// TIA Portal project "tram_2_full_V16" (V16)

(* hardware
DEVICE "S7-1200 station_1"  S7-1200 Station
   slot 0: "Rack_0"  S7-1200 Rack  Rack  V1.0
   slot 1: "PLC_1"  CPU 1214C DC/DC/DC  6ES7 214-1AG40-0XB0  V4.1
   slot 2: "DQ 8xRelay_1"  SM 1222 DQ8 x relay  6ES7 222-1HF32-0XB0  V2.0
DEVICE "HMI_1"  KTP400 Basic PN
   slot 0: "HMI_1"  KTP400 Basic PN  6AV2 123-2DB03-0AX0  15.0.0.0
   slot 1: "HMI_RT_1"  KTP400 Basic PN  6AV2 123-2DB03-0AX0  15.0.0.0
   slot 5: "HMI_1.IE_CP_1"  PROFINET Interface  15.0.0.0
      slot 1: "PROFINET Interface_1"  PROFINET Interface
         slot 1: "Port_1"  Port
*)

// ===== PLC "PLC_1"  CPU 1214C DC/DC/DC =====

VAR_GLOBAL   // PLC tag table "Default tag table"
   "Start" AT %I0.1 : Bool;
   "CylinderB" AT %Q9.6 : Bool;
   "Gripper" AT %Q9.5 : Bool;
   "Arm+" AT %Q9.4 : Bool;
   "Stop" AT %I0.2 : Bool;
   "Arm-" AT %Q9.3 : Bool;
   "CylinderA-" AT %Q9.2 : Bool;
   "CylinderA+" AT %Q9.7 : Bool;
   "Tag_1" AT %M0.1 : Bool;
   "Timer1" AT %MD0 : DWord;
   "LQ2" AT %I0.6 : Bool;
   "SQ3" AT %I0.7 : Bool;
   "Tag_2" AT %M0.2 : Bool;
   "Timer2" AT %MD4 : DWord;
   "Tag_3" AT %M0.3 : Bool;
   "Tag_4" AT %M0.4 : Bool;
   "Tag_5" AT %M1.1 : Bool;
   "Tag_6" AT %M0.7 : Bool;
   "Tag_7" AT %M1.4 : Bool;
   "LQ1" AT %I0.5 : Bool;
   "Tag_8" AT %Q9.0 : Bool;
   "Tag_9" AT %Q9.1 : Bool;
   "Timer4" AT %MD10 : DWord;
   "Timer5" AT %MD14 : DWord;
   "Tag_10" AT %Q0.1 : Bool;
   "Tag_11" AT %Q0.2 : Bool;
   "Tag_12" AT %M0.5 : Bool;
   "MemoryStop" AT %Q0.3 : Bool;
   "Tag_13" AT %Q0.4 : Bool;
   "Tag_14" AT %M4.5 : Bool;
END_VAR

// folder: System blocks/Program resources

DATA_BLOCK "T1"   // DB1
{ S7_Optimized_Access := 'TRUE' }
AUTHOR : Simatic
FAMILY : IEC
NAME : IEC_TMR
VERSION : 1.0
// stored: InstanceOfName IEC_TIMER
"IEC_TIMER"
BEGIN
END_DATA_BLOCK

DATA_BLOCK "T4"   // DB3
{ S7_Optimized_Access := 'TRUE' }
AUTHOR : Simatic
FAMILY : IEC
NAME : IEC_TMR
VERSION : 1.0
// stored: InstanceOfName IEC_TIMER
"IEC_TIMER"
BEGIN
END_DATA_BLOCK

// folder: (top level)

ORGANIZATION_BLOCK "Main"   // OB1, LAD, ProgramCycle
TITLE = "Main Program Sweep (Cycle)"
{ S7_Optimized_Access := 'TRUE' }
VERSION : 0.1
   VAR_INPUT
      Initial_Call : Bool;   // Initial call of this OB
      Remanence : Bool;   // =True, if remanent data are available
   END_VAR
   VAR_TEMP   // added for the SCL form of the ladder/FBD networks
      _w1 : Bool;
   END_VAR
BEGIN

REGION Network 1
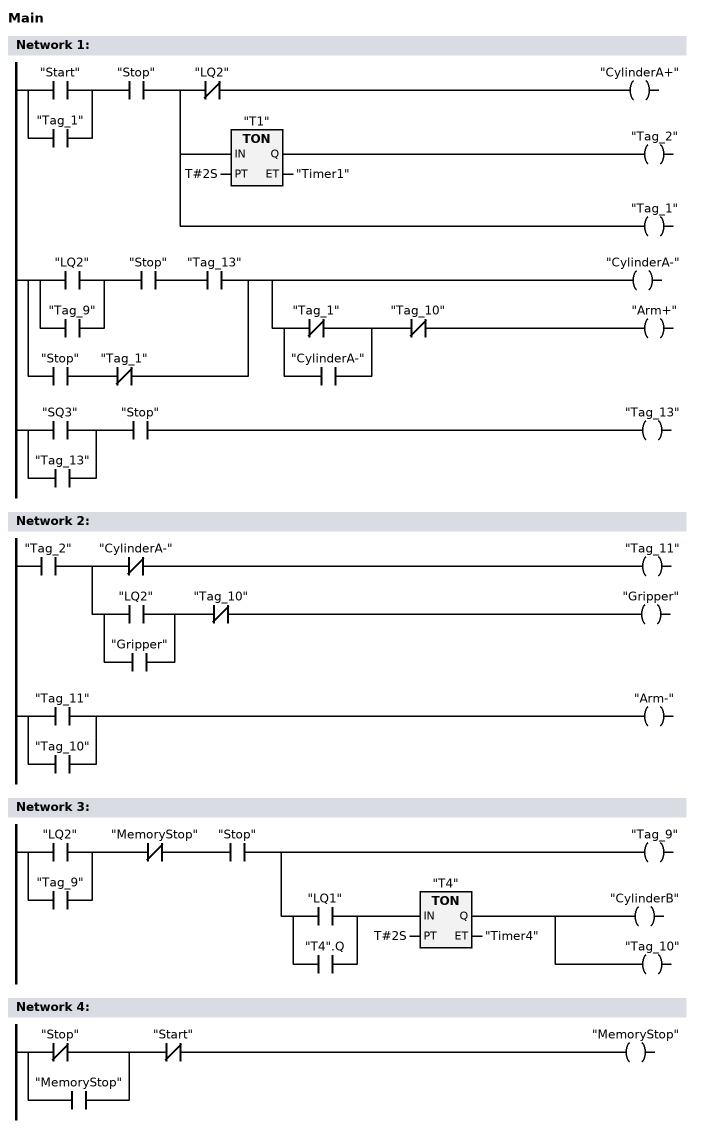
   #_w1 := ("Start" OR "Tag_1") AND "Stop";
   "CylinderA+" := #_w1 AND NOT "LQ2";
   "T1".TON(IN := #_w1, PT := T#2S, ET => "Timer1");
   "Tag_2" := "T1".Q;
   "Tag_1" := #_w1;
   "CylinderA-" := (("LQ2" OR "Tag_9") AND "Stop" AND "Tag_13") OR ("Stop" AND NOT "Tag_1");
   "Arm+" := "CylinderA-" AND (NOT "Tag_1" OR "CylinderA-") AND NOT "Tag_10";
   "Tag_13" := ("SQ3" OR "Tag_13") AND "Stop";
END_REGION

REGION Network 2
   RUNG wire#powerrail
      Contact( "Tag_2" )
      wire#w1
      I_Contact( "CylinderA-" )
      Coil( "Tag_11" )
   END_RUNG
   RUNG wire#w1
      Contact( "LQ2" )
      wire#w2
      I_Contact( "Tag_10" )
      Coil( "Gripper" )
   END_RUNG
   RUNG wire#w1
      Contact( "Gripper" )
   END_RUNG wire#w2
   RUNG wire#powerrail
      Contact( "Tag_11" )
      wire#w3
      Coil( "Arm-" )
   END_RUNG
   RUNG wire#powerrail
      Contact( "Tag_10" )
   END_RUNG wire#w3
   // the same network as SCL:
   "Tag_11" := "Tag_2" AND NOT "CylinderA-";
   "Gripper" := "Tag_2" AND ("LQ2" OR "Gripper") AND NOT "Tag_10";
   "Arm-" := "Tag_11" OR "Tag_10";
END_REGION

REGION Network 3
   "Tag_9" := ("LQ2" OR "Tag_9") AND NOT "MemoryStop" AND "Stop";
   "T4".TON(IN := "Tag_9" AND ("LQ1" OR "T4".Q), PT := T#2S, ET => "Timer4");
   "CylinderB" := "T4".Q;
   "Tag_10" := "T4".Q;
END_REGION

REGION Network 4
   RUNG wire#powerrail
      I_Contact( "Stop" )
      wire#w1
      I_Contact( "Start" )
      Coil( "MemoryStop" )
   END_RUNG
   RUNG wire#powerrail
      Contact( "MemoryStop" )
   END_RUNG wire#w1
   // the same network as SCL:
   "MemoryStop" := (NOT "Stop" OR "MemoryStop") AND NOT "Start";
END_REGION
END_ORGANIZATION_BLOCK

(* ===== HMI "HMI_RT_1" =====
system functions are stored by id; their names below are inferred from use

HMI tags "Default tag table"
   "Tag_ScreenNumber" : UInt, internal

Template "Template_1" 480x272
   Button "Exit" at 388,227 size 63x44; TextOff 'Exit'; PictureOff "ExitRuntime_KTP400_Basic_PN_TR"; PictureOn "ExitRuntime_KTP400_Basic_PN_TR"
      on Release: StopRuntime(0)
   Button "Template_Button" at 268,227 size 63x44; TextOff 'Text'
   Button "Alarms" at 148,227 size 63x44; TextOff 'Alarms'; PictureOff "AlarmDisplay_KTP400_Basic_PN_TR"; PictureOn "AlarmDisplay_KTP400_Basic_PN_TR"
      on Release: function_ef3f5d25("Alarm window_Unacknowledged", -1)
   Button "Start screen" at 28,227 size 63x44; TextOff 'Start screen'; PictureOff "NavigateHome_KTP400_Basic_PN_TR"; PictureOn "NavigateHome_KTP400_Basic_PN_TR"
      on Release: ActivateScreen("Root screen", 0)
   SymbolicIOField "Symbolic_IO_Field_Screen" at 82,8 size 311x29; TextOff '0'; TextOn '1'; TextList "TextList_ScreenNames"
      ProcessValue <- "Tag_ScreenNumber"
      on Change: ActivateScreenByNumber("Tag_ScreenNumber", 0)
   DateTimeField "HmiScreenItemData" at 395,22 size 85x22
   DateTimeField "HmiScreenItemData_1" at 395,0 size 85x22
   GraphicView "Logo" at 0,0 size 80x45; Picture "Logo of HMI_1"

screen "Root screen" 480x272, template "Template_1"
   on GenerateScreen: SetTag("Tag_ScreenNumber", 1)
   TextField "HmiScreenItemData" at 48,122 size 384x22; Text 'Welcome to HMI_1 (KTP400 Basic+ PN)!'
*)